(* IEC 61131-3 sources: CS_4_Aufzugsteuerung/src/Stations/CP112/Steuerung/Class/clsAufzugmodul, 1 file *)

(* ---- clsAufzugmodul.st ---- *)
(*!
<Class
	Name               = "clsAufzugmodul"
	Revision           = "0.0"
	RealtimeTask       = "true"
	CyclicTask         = "false"
	DefCyclictime      = "1 ms"
	BackgroundTask     = "false"
	Sigmatek           = "false"
	OSInterface        = "false"
	HighPriority       = "false"
	Automatic          = "false"
	UpdateMode         = "Prescan"
	SharedCommandTable = "true"
	Objectsize         = "(284,120)">
	<Channels>
		<Server Name="ClassSvr" Visualized="false" Initialize="false" WriteProtected="true" Retentive="false"/>
		<Client Name="cAnforderung" Required="true" Internal="false"/>
		<Client Name="cAntriebAufzug" Required="true" Internal="false"/>
		<Client Name="cAntriebTuer" Required="true" Internal="false"/>
		<Client Name="cEMG_Stop" Required="true" Internal="false"/>
		<Client Name="cEtagestatus" Required="true" Internal="false"/>
		<Client Name="cTimerOffen" Required="true" Internal="false"/>
		<Client Name="cTuerstatus" Required="true" Internal="false"/>
		<Client Name="cZeitOffen" Required="false" Internal="false"/>
	</Channels>
</Class>
*)
clsAufzugmodul : CLASS
	TYPE
	  Schritkette :
	  (
	    Initialisierung:=0,
	    Fahranforderung:=10,
	    FahrrichtungSuchen:=20,
	    InitFahrtnachOben:=30,
	    Hochfahrt:=31,
	    EtagenOben:=32,
	    TuerOeffnen:=33,
	    TuerSchliessen,
	    InitFahrtnachUnten:=40,
	    Unterfahrt:=41,
	    EtageUnten:=42,
	    NotAus
	  )$UDINT;
	END_TYPE
  //Servers:
	ClassSvr 	: SvrChCmd_DINT;
  //Clients:
	cEtagestatus 	: CltChCmd_clsEtagenSensorik;
	cTuerstatus 	: CltChCmd_clsTuerSensorik;
	cAntriebAufzug 	: CltChCmd_clsAntrieb;
	cAntriebTuer 	: CltChCmd_clsAntrieb;
	cAnforderung 	: CltChCmd_clsHauptablauf;
	cTimerOffen 	: CltChCmd_clsTimer;
	cZeitOffen 	: CltCh_UDINT;
	cEMG_Stop 	: CltChCmd_clsEmgStop_1;
  //Variables:
		iStep 	: Schritkette;
		iAktEtage 	: DINT;
		xZielOben 	: BOOL;
		xZielUnten 	: BOOL;
  //Functions:

	FUNCTION VIRTUAL GLOBAL RtWork
		VAR_INPUT
			EAX 	: UDINT;
		END_VAR
		VAR_OUTPUT
			state (EAX) 	: UDINT;
		END_VAR;
  //Tables:
	FUNCTION @STD
		VAR_OUTPUT
			ret_code	: CONFSTATES;
		END_VAR;
	FUNCTION GLOBAL TAB @CT_;
END_CLASS;

#pragma usingLtd clsAntrieb
#pragma usingLtd clsEmgStop_1
#pragma usingLtd clsEtagenSensorik
#pragma usingLtd clsHauptablauf
#pragma usingLtd clsTimer
#pragma usingLtd clsTuerSensorik

FUNCTION VIRTUAL GLOBAL clsAufzugmodul::RtWork
	VAR_INPUT
		EAX 	: UDINT;
	END_VAR
	VAR_OUTPUT
		state (EAX) 	: UDINT;
	END_VAr

  //Notaus zustand
  IF cEMG_Stop.EmgStop() THEN
    iStep := NotAus;
  END_IF;

  // Parameter lesen
  cEMG_Stop := cEMG_Stop.Read();
  cZeitOffen := cZeitOffen.Read();

  // Aktuelle Etage lesen
  iAktEtage := cEtagestatus.AktEtage();

  CASE iStep OF

  Initialisierung:

      cAntriebAufzug.Fahrt(xDir := FALSE, xStart := FALSE);
      cAntriebTuer.Fahrt(xDir := FALSE, xStart := FALSE);

      iStep := Fahranforderung;

  Fahranforderung:

      IF cAnforderung.Anf0(xIn := FALSE) OR
         cAnforderung.Anf1(xIn := FALSE) OR
         cAnforderung.Anf2(xIn := FALSE) OR
         cAnforderung.Anf3(xIn := FALSE) THEN

          iStep := FahrrichtungSuchen;

      ELSIF cAnforderung.TuerAuf() THEN // falls jemand im Lift bleibt und nach schliessung aufmachen will
         iStep := TuerOeffnen;
      END_IF;

  FahrrichtungSuchen:

      xZielOben := FALSE;
      xZielUnten := FALSE;

      CASE iAktEtage OF

          0:
              IF cAnforderung.Anf1(xIn := FALSE) OR
                 cAnforderung.Anf2(xIn := FALSE) OR
                 cAnforderung.Anf3(xIn := FALSE) THEN
                  xZielOben := TRUE;
              END_IF;

          1:
              IF cAnforderung.Anf2(xIn := FALSE) OR
                 cAnforderung.Anf3(xIn := FALSE) THEN
                  xZielOben := TRUE;
              END_IF;

              IF cAnforderung.Anf0(xIn := FALSE) THEN
                  xZielUnten := TRUE;
              END_IF;

          2:

              IF cAnforderung.Anf3(xIn := FALSE) THEN
                  xZielOben := TRUE;
              END_IF;

              IF cAnforderung.Anf0(xIn := FALSE) OR
                 cAnforderung.Anf1(xIn := FALSE) THEN
                  xZielUnten := TRUE;
              END_IF;

          3:

              IF cAnforderung.Anf0(xIn := FALSE) OR
                 cAnforderung.Anf1(xIn := FALSE) OR
                 cAnforderung.Anf2(xIn := FALSE) THEN
                  xZielUnten := TRUE;
              END_IF;

      END_CASE;

      IF xZielOben THEN
          iStep := InitFahrtnachOben;

      ELSIF xZielUnten THEN
          iStep := InitFahrtnachUnten;

      ELSE
          iStep := TuerOeffnen; //wenn die Anforderung auf der bereits stehenden Etage kommt,oeffnen
      END_IF;

  InitFahrtnachOben:

      IF cTuerstatus.istzu() THEN

          cAntriebTuer.Fahrt(xDir := FALSE, xStart := FALSE);
          iStep := Hochfahrt;

      ELSIF cAnforderung.TuerAuf() THEN

          iStep := TuerOeffnen;

      ELSE

          cTuerstatus.zu(); // Simulation
          cAntriebTuer.Fahrt(xDir := TRUE, xStart := TRUE); // Tür schliessen

      END_IF;

  Hochfahrt:

      cEtagestatus.hoch();
      cAntriebAufzug.Fahrt(xDir := TRUE, xStart := TRUE);

      IF cEtagestatus.erreicht() THEN
          cAntriebAufzug.Fahrt(xDir := TRUE, xStart := FALSE);
          iStep := EtagenOben;
      END_IF;

  EtagenOben:

      iAktEtage := cEtagestatus.AktEtage();

      IF (cAnforderung.Anf0(xIn := FALSE) AND (iAktEtage = 0)) OR
         (cAnforderung.Anf1(xIn := FALSE) AND (iAktEtage = 1)) OR
         (cAnforderung.Anf2(xIn := FALSE) AND (iAktEtage = 2)) OR
         (cAnforderung.Anf3(xIn := FALSE) AND (iAktEtage = 3)) THEN

          cAntriebAufzug.Fahrt(xDir := TRUE, xStart := FALSE);
          iStep := TuerOeffnen;

      ELSE

          iStep := Hochfahrt;

      END_IF;

  InitFahrtnachUnten:

      IF cTuerstatus.istzu() THEN

          cAntriebTuer.Fahrt(xDir := FALSE, xStart := FALSE);
          iStep := Unterfahrt;

      ELSIF cAnforderung.TuerAuf() THEN

          iStep := TuerOeffnen;

      ELSE

          cTuerstatus.zu(); // Simulation
          cAntriebTuer.Fahrt(xDir := TRUE, xStart := TRUE); // Tür schliessen

      END_IF;

  Unterfahrt:

      cEtagestatus.runter();
      cAntriebAufzug.Fahrt(xDir := FALSE, xStart := TRUE);

      IF cEtagestatus.erreicht() THEN
          cAntriebAufzug.Fahrt(xDir := FALSE, xStart := FALSE);
          iStep := EtageUnten;
      END_IF;

  EtageUnten:

      iAktEtage := cEtagestatus.AktEtage();

      IF (cAnforderung.Anf0(xIn := FALSE) AND (iAktEtage = 0)) OR
         (cAnforderung.Anf1(xIn := FALSE) AND (iAktEtage = 1)) OR
         (cAnforderung.Anf2(xIn := FALSE) AND (iAktEtage = 2)) OR
         (cAnforderung.Anf3(xIn := FALSE) AND (iAktEtage = 3)) THEN

          cAntriebAufzug.Fahrt(xDir := FALSE, xStart := FALSE);
          iStep := TuerOeffnen;

      ELSE

          iStep := Unterfahrt;

      END_IF;

  TuerOeffnen:

      cTuerstatus.auf(); // Simulation
      cAntriebTuer.Fahrt(xDir := FALSE, xStart := TRUE); // Tür öffnen

      IF cTuerstatus.istauf() THEN

          cAntriebTuer.Fahrt(xDir := FALSE, xStart := FALSE);

          IF NOT cTimerOffen.running() THEN
              cTimerOffen.start(_time := cZeitOffen);
          END_IF;

      END_IF;

      IF cTimerOffen.elapsed() OR cAnforderung.TuerZu() THEN

          cTimerOffen.reset();
          iStep := TuerSchliessen;

      END_IF;

 TuerSchliessen:

    IF cAnforderung.TuerAuf() THEN

        cAntriebTuer.Fahrt(xDir := TRUE, xStart := FALSE);
        iStep := TuerOeffnen;

    ELSE

        cTuerstatus.zu(); // Simulation
        cAntriebTuer.Fahrt(xDir := TRUE, xStart := TRUE); // Tür schliessen

        IF cTuerstatus.istzu() THEN

            cAntriebTuer.Fahrt(xDir := TRUE, xStart := FALSE);

            iAktEtage := cEtagestatus.AktEtage();

            IF iAktEtage = 0 THEN
                cAnforderung.Anf0(xIn := TRUE);

            ELSIF iAktEtage = 1 THEN
                cAnforderung.Anf1(xIn := TRUE);

            ELSIF iAktEtage = 2 THEN
                cAnforderung.Anf2(xIn := TRUE);

            ELSIF iAktEtage = 3 THEN
                cAnforderung.Anf3(xIn := TRUE);

            END_IF;

            iStep := Initialisierung;

        END_IF;

    END_IF;

  NotAus:
    cAntriebAufzug.NotAus(xIn:=TRUE);
    cAntriebTuer.NotAus(xIn:=TRUE);

    IF NOT cEMG_Stop.EmgStop()  THEN
      cAntriebAufzug.NotAus(xIn:=FALSE);
      cAntriebTuer.NotAus(xIn:=FALSE);
      iStep := Initialisierung;
    END_IF;

  END_CASE;

 cEMG_Stop:= 1;

	state := READY;

END_FUNCTION
